FUNCTION_BLOCK SPLIT_AQ_INTO_AX (* splits a 2-bit AQ adapter into 2 AX (BOOL) adapters *)
  (* Standard: 61499-2; Description: Copyright (c) 2026 Meisterschulen am Ostbahnhof SPDX-License-Identifier: EPL-2.0 *)
  (* Version 1.0, 2026-05-16, Franz Höpfinger, Meisterschulen am Ostbahnhof, Initial Version *)
  PACKAGE adapter::splitting;
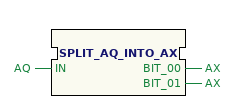
  SOCKETS
    IN : adapter::types::unidirectional::AQ; (* AQ Input *)
  END_SOCKETS
  PLUGS
    BIT_00 : adapter::types::unidirectional::AX; (* Bit 0 *)
    BIT_01 : adapter::types::unidirectional::AX; (* Bit 1 *)
  END_PLUGS
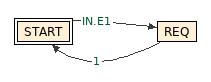
  EC_STATES
    START;
    REQ;
  END_STATES
  EC_TRANSITIONS
    START TO REQ := IN.E1;
    REQ TO START := 1;
  END_TRANSITIONS
  ALGORITHM REQ IN ST:
BIT_00.D1 := IN.D1.%X0;
BIT_01.D1 := IN.D1.%X1;
BIT_00.E1();
BIT_01.E1();
  END_ALGORITHM
END_FUNCTION_BLOCK
(* other elements stored in the file *)
(* Algorithm Name=REQ *)
